INTERFACE I_Cylinder EXTENDS I_ActuatorWorkBase

METHOD enable : BOOL //Result value = successful execution of desired action 
VAR_INPUT
	IN							:	BOOL; //TRUE = to Work pos / FLASE = to base pos
END_VAR
END_METHOD

{attribute 'monitoring' := 'call'}
PROPERTY PUBLIC inError : Bool
GET
END_GET
END_PROPERTY

{attribute 'monitoring' := 'call'}
PROPERTY isBusy : BOOL
GET
END_GET
END_PROPERTY

{attribute 'monitoring' := 'call'}
PROPERTY isInBasePos : BOOL
GET
END_GET
END_PROPERTY

{attribute 'monitoring' := 'call'}
PROPERTY isInWorkPos : BOOL
GET
END_GET
END_PROPERTY

METHOD PUBLIC moveToBasePos : BOOL //Return = Done -> InBasePos
END_METHOD

METHOD PUBLIC moveToWorkPos : BOOL //Return = Done -> InWorkPos
END_METHOD

{attribute 'monitoring' := 'call'}
PROPERTY noFeed : BOOL
GET
END_GET
END_PROPERTY

{attribute 'monitoring' := 'call'}
PROPERTY PUBLIC rCylinder : REFERENCE TO Cylinder
GET
END_GET
END_PROPERTY

{attribute 'monitoring' := 'call'}
PROPERTY simulation : BOOL
GET
END_GET
SET
END_SET
END_PROPERTY

METHOD PUBLIC switchOff : BOOL
VAR_INPUT
END_VAR
END_METHOD

END_INTERFACE

(* stored: Version 1.1.0.1, ProductVersion 3.1.4024.13
   Itf I_Cylinder: Id {4d2373c8-2760-49ad-87af-d4082e0bb0ba}
   Method enable: Id {e4f0239a-dfff-456c-9610-8c975276794c}
   Property inError: Id {2a3db1e8-9167-420f-9c58-a14c446a0406}
   Get Get: Id {637fc8c7-88ff-41f0-88b9-113a7e814405}
   Property isBusy: Id {d2bfd107-8d51-4229-bcc3-42f04887b647}
   Get Get: Id {2f3ccf62-bb7e-42e7-bb50-da66199bf6c2}
   Property isInBasePos: Id {144ba97a-dafe-4a4d-b244-eff50927a481}
   Get Get: Id {2f624f26-ec4c-4240-9be8-67ff899ff7ed}
   Property isInWorkPos: Id {2d9eb0a7-3b1d-4f8a-9efd-2dae1699b26f}
   Get Get: Id {e479d18e-d6e9-4b93-a58a-01040a2c84d7}
   Method moveToBasePos: Id {3c4995cb-c8da-43d1-bebb-265d8ef4ecce}
   Method moveToWorkPos: Id {5bdeb475-d97a-434f-8399-4fa795a3d6a6}
   Property noFeed: Id {7ed343f7-7775-43c9-b6d3-64d82bac56d9}
   Get Get: Id {d23d00d7-e588-43e0-8191-aa7f20c3cd6b}
   Property rCylinder: Id {dad555d2-b66e-4daf-bb58-2fc8f90962eb}
   Get Get: Id {23918dde-c9df-4d02-9c90-79cc2a49d4d7}
   Property simulation: Id {b63ad6e8-a595-4c2c-beb8-b12826329149}
   Get Get: Id {fb0211f2-a8c5-41a0-b9f7-f95a7fd07d66}
   Set Set: Id {f5b13c02-fd36-4547-82e4-307be261014b}
   Method switchOff: Id {fdb6901a-99c7-489f-8d3c-2770508a80b9} *)
